{attribute 'linkalways'} 
{attribute 'no_explicit_call' := 'This FB is a CLASS and must be accessed using methods or properties'}
{attribute 'enable_dynamic_creation'}
FUNCTION_BLOCK _Array0to3OfUINT EXTENDS ArrayDatatypeBase_1D
VAR CONSTANT
	lBound : DINT := 0;
	uBound : DINT := 3;
END_VAR
VAR
	localData : ARRAY [lBound..uBound] OF UINT;
	activeData : REFERENCE TO ARRAY [lBound..uBound] OF UINT REF= localData;
	elements : ARRAY [lBound..uBound] OF _UINT(0);
	baseType : _UINT(0);
END_VAR

PROPERTY PUBLIC Address : PVOID
GET
Address := ADR(activeData);
END_GET
END_PROPERTY

PROPERTY PUBLIC BaseDatatype : I_Datatype
GET
BaseDatatype := baseType;
END_GET
END_PROPERTY

METHOD PUBLIC ClearReference
VAR_INPUT
END_VAR
activeData REF= localData;
SetElementReference();
END_METHOD

METHOD PUBLIC Clone : I_Datatype
VAR
    pClone : POINTER TO _Array0to3OfUINT;
END_VAR
pClone := __NEW(_Array0to3OfUINT());
pClone^.Value := Value;
Clone := pClone^;
END_METHOD

METHOD FB_init : BOOL
VAR_INPUT
	bInitRetains : BOOL; // if TRUE, the retain variables are initialized (warm start / cold start)
	bInCopyCode : BOOL;  // if TRUE, the instance afterwards gets moved into the copy code (online change)
END_VAR
SetElementReference();
END_METHOD

METHOD PUBLIC MakeReferenceTo
VAR_INPUT
	ReferenceTarget : REFERENCE TO ARRAY [lBound..uBound] OF UINT;
END_VAR
activeData REF= ReferenceTarget;
SetElementReference();
END_METHOD

METHOD PROTECTED OnSerializeArrayValues
VAR_INPUT
	Serializer : I_Serializer;
END_VAR
VAR
	i : DINT;
END_VAR
FOR i := lBound TO uBound DO
	elements[i].SerializeWith(Serializer);
END_FOR
END_METHOD

METHOD PROTECTED SetElementReference
VAR_INPUT
END_VAR
VAR
	i : DINT;
END_VAR
FOR i := lBound TO uBound DO
	elements[i].MakeReferenceTo(activeData[i]);
END_FOR
END_METHOD

PROPERTY PUBLIC Size : UDINT
GET
Size := SIZEOF(activeData);
END_GET
END_PROPERTY

METHOD PROTECTED TryDeserializeArrayValues : BOOL
VAR_INPUT
	Deserializer : I_Deserializer;
	Feedback : I_DeserializerFeedback;
END_VAR
VAR
	enumerator : I_DeserializerArrayForwardEnumerator;
	i : DINT;
END_VAR
enumerator := Deserializer.GetArrayEnumerator();
i := lBound;

WHILE enumerator.MoveNext() AND i <= uBound DO
	
	IF NOT elements[i].TryDeserializeFrom(enumerator.Current, Feedback) THEN
		EXIT;
	END_IF
	i := i + 1;

END_WHILE
enumerator.Dispose();
END_METHOD

METHOD PUBLIC TryGetElementAsDatatypeByIndex : BOOL
VAR_INPUT
	Index : DINT;
	Destination : REFERENCE TO I_Datatype;
END_VAR
IF Index < lbound OR Index > ubound THEN
	RETURN;
END_IF

Destination := elements[Index];
TryGetElementAsDatatypeByIndex := TRUE;
END_METHOD

METHOD PUBLIC TryGetLowerBound : BOOL
VAR_INPUT
	Dimention : UDINT;
	Destination : REFERENCE TO DINT;
END_VAR
IF Dimention = 1 THEN
	Destination := lBound;
	TryGetLowerBound := TRUE;
END_IF
END_METHOD

METHOD PUBLIC TryGetUpperBound : BOOL
VAR_INPUT
	Dimention : UDINT;
	Destination : REFERENCE TO DINT;
END_VAR
IF Dimention = 1 THEN
	Destination := uBound;
	TryGetUpperBound := TRUE;
END_IF
END_METHOD

METHOD TryMakeReferenceTo : BOOL
VAR_INPUT
	Target : I_Datatype;
END_VAR
VAR
	pTargetData : POINTER TO ARRAY [lBound..uBound] OF UINT;
END_VAR
IF NOT IsEquivalentTo(Target) THEN
	RETURN;
END_IF

pTargetData := Target.Address;
activeData REF= pTargetData^;
SetElementReference();
TryMakeReferenceTo := TRUE;
END_METHOD

PROPERTY PUBLIC Value : REFERENCE TO ARRAY [lBound..uBound] OF UINT;
GET
Value ref= activeData;
END_GET
END_PROPERTY

END_FUNCTION_BLOCK

(* stored: Version 1.1.0.1, ProductVersion 3.1.4024.13
   POU _Array0to3OfUINT: Id {c3a26628-c459-031d-33a9-3fffa547078d}, SpecialFunc None
   Folder Core: Id {1cf9d0da-516d-027d-0c8c-9f7d6d17850c}
   Folder Constructor: Id {6671630f-0467-0309-0c5e-a26a853ba4b8}
   Folder Protected: Id {10bbf441-6d6b-0527-2ea7-285db25f4643}
   Folder Customize: Id {59191baf-95ed-0bf6-1c02-12e0bdd076a3}
   Property Address: Id {897c41a9-5f73-00a7-1b69-8a5d80bb0931}
   Get Get: Id {de4755dc-0746-0414-1b5d-efe53a41c6bb}
   Property BaseDatatype: Id {88bd5b50-a7d2-0cd1-1c0c-327dc74fedb3}
   Get Get: Id {b5cfd9f8-264a-0d83-1560-d70e5b897bcd}
   Method ClearReference: Id {3b651948-f250-0f77-0b8f-61f541e9cb99}
   Method Clone: Id {663d0f86-5953-05db-2ad4-b2f2ae96e4b2}
   Method FB_init: Id {cfec4b60-c44e-0d16-3d7b-38937efb07fd}
   Method MakeReferenceTo: Id {4489b418-9725-0a0e-07b9-2e904ac3cecf}
   Method OnSerializeArrayValues: Id {17bc89e8-5601-04f1-3918-0c41d5c6d658}
   Method SetElementReference: Id {27a63faf-96e0-0525-34a7-2d6edf2f1820}
   Property Size: Id {1b7a7e0e-1e0e-00df-04f0-e7977146ccf0}
   Get Get: Id {1d9ee7fb-c894-0ce4-34cb-d25b8df0d9df}
   Method TryDeserializeArrayValues: Id {ca919786-6c4b-0657-3a9d-3923935c4f47}
   Method TryGetElementAsDatatypeByIndex: Id {88aba39d-71ba-0994-00f2-133f0e081136}
   Method TryGetLowerBound: Id {407e92fc-a199-0d1d-33a4-653c36e1be31}
   Method TryGetUpperBound: Id {41097f97-cb99-04bc-0c33-c03beb59b43f}
   Method TryMakeReferenceTo: Id {0092f664-e65c-0a74-2acd-19af5fed976b}
   Property Value: Id {8b19877f-4ed5-0583-23d0-d8b9fd791b7d}
   Get Get: Id {7ba79c2c-f684-0e75-10de-ea6c9a45153f} *)
